Fanuc KAREL source: kt00859.KL

-- PROVISIONAL review KL for V1013-1; original PC SHA256 0491ab513b6da8afbf32b4268a0a5229b792efceda6742d995ed12b7eb00a730
-- Incomplete behavior may be omitted. Consult companion uncertainty JSON. Do not deploy.
PROGRAM KT00859
%NOLOCKGROUP
VAR
  R1 : REAL
  R2 : REAL
  OUT : REAL
BEGIN
  -- UNRESOLVED_PC offsets 5-16; opcodes 2E,23
  -- UNRESOLVED_PC offsets 21-32; opcodes 2E,23
  -- UNRESOLVED_PC offsets 37-48; opcodes 2E,23
  -- UNRESOLVED_PC offsets 53-64; opcodes 2E,23
  -- UNRESOLVED_PC offsets 69-85; opcodes 27,22,76,64,23
  -- UNRESOLVED_PC offsets 90-94; opcodes 7F
END KT00859
